% RSLogix 500 project ESTACION3.RSS, saved by version 8.40.00.08 %
PROJECT "UNTITLED"    % processor: MicroLogix 1500 %

PROGRAM FILES
  LAD 2   19 rungs

DATA FILES
  O0 OUTPUT  4 elements
  I1 INPUT  4 elements
  S2 STATUS  66 elements
  B3 BINARY  1 elements
  T4 TIMER  4 elements
  C5 COUNTER  1 elements
  R6 CONTROL  1 elements
  N7 INTEGER  1 elements
  F8 FLOAT  1 elements

LADDER 2
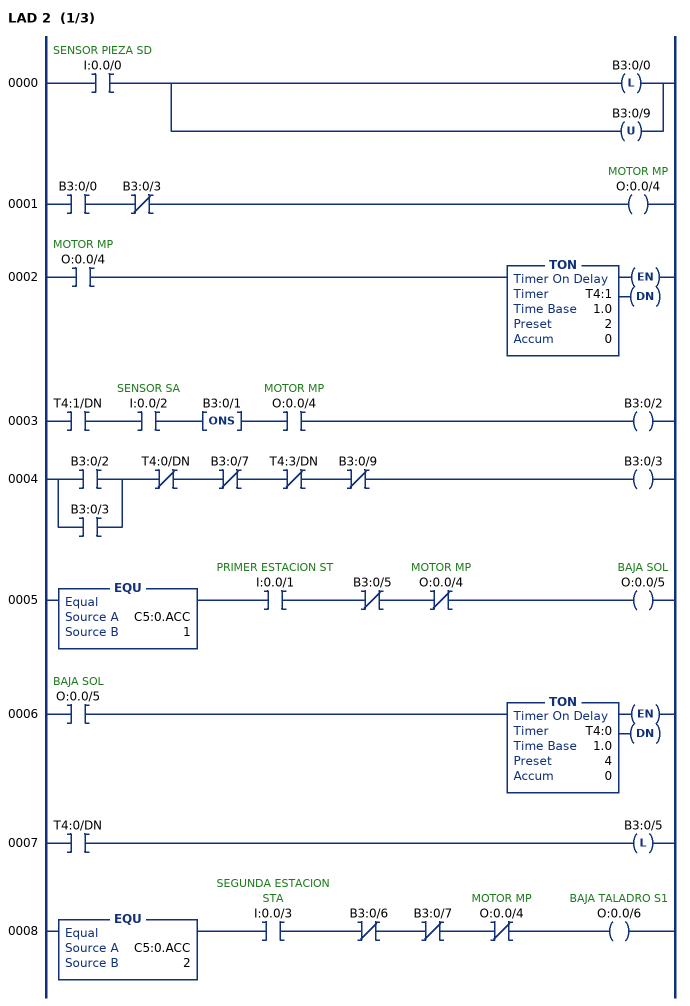
% Rung: 0 %
SOR XIC I:0.0/0 BST OTL B3:0/0 NXB OTU B3:0/9 BND EOR
%   I:0.0/0  "SENSOR PIEZA SD" %
% Rung: 1 %
SOR XIC B3:0/0 XIO B3:0/3 OTE O:0.0/4 EOR
%   O:0.0/4  "MOTOR MP" %
% Rung: 2 %
SOR XIC O:0.0/4 TON T4:1 1.0 2 0 EOR
%   O:0.0/4  "MOTOR MP" %
% Rung: 3 %
SOR XIC T4:1/DN XIC I:0.0/2 ONS B3:0/1 XIC O:0.0/4 OTE B3:0/2 EOR
%   I:0.0/2  "SENSOR SA" %
%   O:0.0/4  "MOTOR MP" %
% Rung: 4 %
SOR BST XIC B3:0/2 NXB XIC B3:0/3 BND XIO T4:0/DN XIO B3:0/7 XIO T4:3/DN XIO B3:0/9 OTE B3:0/3 EOR
% Rung: 5 %
SOR EQU C5:0.ACC 1 XIC I:0.0/1 XIO B3:0/5 XIO O:0.0/4 OTE O:0.0/5 EOR
%   I:0.0/1  "PRIMER ESTACION ST" %
%   O:0.0/4  "MOTOR MP" %
%   O:0.0/5  "BAJA SOL" %
% Rung: 6 %
SOR XIC O:0.0/5 TON T4:0 1.0 4 0 EOR
%   O:0.0/5  "BAJA SOL" %
% Rung: 7 %
SOR XIC T4:0/DN OTL B3:0/5 EOR
% Rung: 8 %
SOR EQU C5:0.ACC 2 XIC I:0.0/3 XIO B3:0/6 XIO B3:0/7 XIO O:0.0/4 OTE O:0.0/6 EOR
%   I:0.0/3  "SEGUNDA ESTACION STA" %
%   O:0.0/4  "MOTOR MP" %
%   O:0.0/6  "BAJA TALADRO S1" %

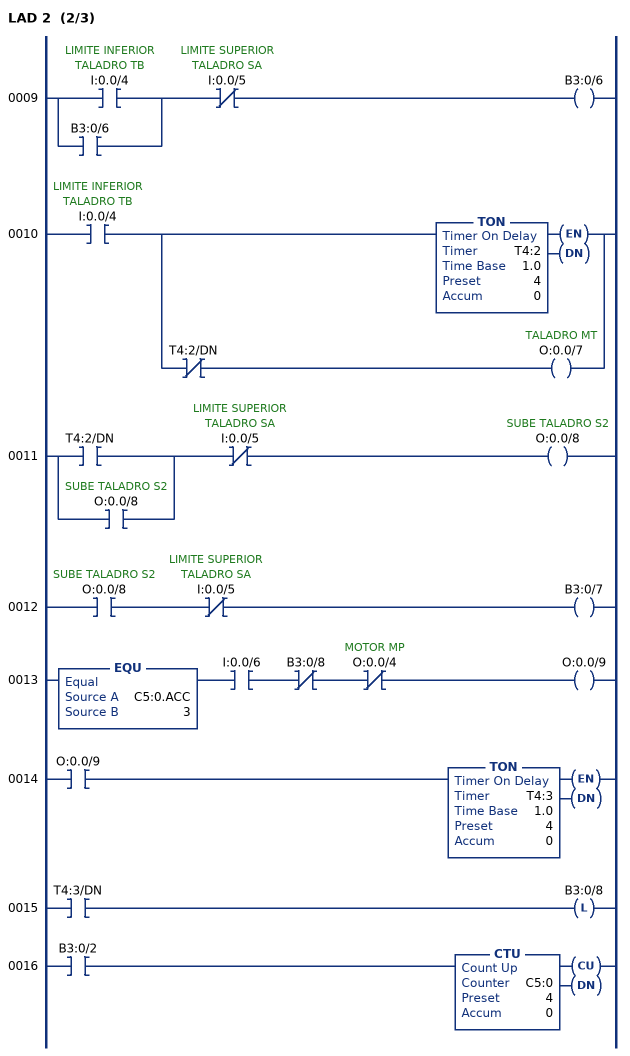
% Rung: 9 %
SOR BST XIC I:0.0/4 NXB XIC B3:0/6 BND XIO I:0.0/5 OTE B3:0/6 EOR
%   I:0.0/4  "LIMITE INFERIOR TALADRO TB" %
%   I:0.0/5  "LIMITE SUPERIOR TALADRO SA" %
% Rung: 10 %
SOR XIC I:0.0/4 BST TON T4:2 1.0 4 0 NXB XIO T4:2/DN OTE O:0.0/7 BND EOR
%   I:0.0/4  "LIMITE INFERIOR TALADRO TB" %
%   O:0.0/7  "TALADRO MT" %
% Rung: 11 %
SOR BST XIC T4:2/DN NXB XIC O:0.0/8 BND XIO I:0.0/5 OTE O:0.0/8 EOR
%   O:0.0/8  "SUBE TALADRO S2" %
%   I:0.0/5  "LIMITE SUPERIOR TALADRO SA" %
% Rung: 12 %
SOR XIC O:0.0/8 XIO I:0.0/5 OTE B3:0/7 EOR
%   O:0.0/8  "SUBE TALADRO S2" %
%   I:0.0/5  "LIMITE SUPERIOR TALADRO SA" %
% Rung: 13 %
SOR EQU C5:0.ACC 3 XIC I:0.0/6 XIO B3:0/8 XIO O:0.0/4 OTE O:0.0/9 EOR
%   O:0.0/4  "MOTOR MP" %
% Rung: 14 %
SOR XIC O:0.0/9 TON T4:3 1.0 4 0 EOR
% Rung: 15 %
SOR XIC T4:3/DN OTL B3:0/8 EOR
% Rung: 16 %
SOR XIC B3:0/2 CTU C5:0 4 0 EOR

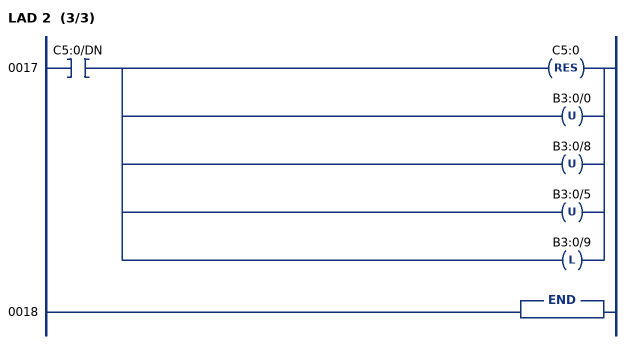
% Rung: 17 %
SOR XIC C5:0/DN BST RES C5:0 NXB BST OTU B3:0/0 NXB BST OTU B3:0/8 NXB BST OTU B3:0/5 NXB OTL B3:0/9 BND BND BND BND EOR
% Rung: 18 %
SOR END EOR

DATA TABLE (non-zero values as saved)
DATA T4
% .PRE .ACC %
% T4:0 % 4 0
% T4:1 % 2 0
% T4:2 % 4 0
% T4:3 % 4 0
DATA C5
% .PRE .ACC %
% C5:0 % 4 0
